// TIA Portal V19 export
FUNCTION_BLOCK "fbGetDiagPnPnCouplerDiag"   // FB1, LAD
{ S7_Optimized_Access := 'TRUE' }
// stored: MemoryReserve 100, SetENOAutomatically false
   VAR_INPUT
      LADDR : HW_ANY;   // Hardware Address of the ~IODevice number
      DebounceTimer : Time := T#3ms;
   END_VAR
   VAR_OUTPUT
      OwnState : UInt;
      SubordinateState : UInt;
      DeviceStatusOk : Bool;
   END_VAR
   VAR
      Diag : DIS;
      Sub { S7_SetPoint := 'True'} : DNN;
      RetValueDiag : Int;
      CntDiagDiag : UInt;
      RetValueSub : Int;
      CntDiagSub : UInt;
      BadStateDebounceTimer : IEC_TIMER;
   END_VAR
   VAR CONSTANT
      "IO Device Mode" : Int := 1;
      "Subordinate device Mode" : Int := 2;
   END_VAR
   VAR_TEMP   // added for the SCL form of the ladder/FBD networks
      _w1 : Bool;
   END_VAR
BEGIN

REGION Network 1: PnPnCoupler Left Get Diag
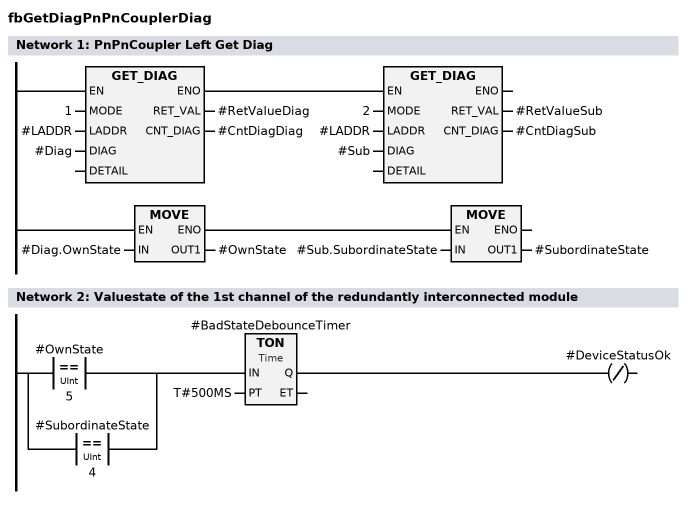
   RUNG wire#powerrail
      GET_DIAG(MODE := 1, LADDR := #LADDR, DIAG := #Diag, DETAIL :=, RET_VAL => #RetValueDiag, CNT_DIAG => #CntDiagDiag)
      GET_DIAG(MODE := 2, LADDR := #LADDR, DIAG := #Sub, DETAIL :=, RET_VAL => #RetValueSub, CNT_DIAG => #CntDiagSub)
   END_RUNG
   RUNG wire#powerrail
      Move(in := #Diag.OwnState, out1 => #OwnState)
      Move(in := #Sub.SubordinateState, out1 => #SubordinateState)
   END_RUNG
   // the same network as SCL:
   #RetValueDiag := GET_DIAG(MODE := 1, LADDR := #LADDR, DIAG := #Diag, CNT_DIAG => #CntDiagDiag, ENO => #_w1);
   IF #_w1 THEN
       #RetValueSub := GET_DIAG(MODE := 2, LADDR := #LADDR, DIAG := #Sub, CNT_DIAG => #CntDiagSub);
   END_IF;
   #OwnState := #Diag.OwnState;
   #SubordinateState := #Sub.SubordinateState;
END_REGION

REGION Network 2: Valuestate of the 1st channel of the redundantly interconnected module
   RUNG wire#powerrail
      { S7_Templates := "SrcType := UInt" } EQ_Contact(in1 := #OwnState, in2 := 5)
      wire#w1
      { S7_Templates := "time_type := Time" } #BadStateDebounceTimer.TON(pt := T#500MS, et =>)
      I_Coil( #DeviceStatusOk )
   END_RUNG
   RUNG wire#powerrail
      { S7_Templates := "SrcType := UInt" } EQ_Contact(in1 := #SubordinateState, in2 := 4)
   END_RUNG wire#w1
   // the same network as SCL:
   #BadStateDebounceTimer.TON(IN := (#OwnState = 5) OR (#SubordinateState = 4), PT := T#500MS);
   #DeviceStatusOk := NOT #BadStateDebounceTimer.Q;
END_REGION
END_FUNCTION_BLOCK
